FUNCTION proj0_TupleStruct_2: BOOL
{ S7_Optimized_Access := 'true' }
    VAR_INPUT
        tuple: TupleStruct_2;
    END_VAR

BEGIN
    proj0_TupleStruct_2 := tuple.field0;
END_FUNCTION
